{attribute 'GeneratedUsingTerminal: EK1122-0000-0018'}
{attribute addProperty BoxType "EK1122-0000-0018"}
{attribute addProperty Id "Beckhoff_EP2xxxsub_EK1100EK1100_1FC0878B2A_0001_EP2001_1000_0016EP2001_C23D36A611A_0002_EP2001_1000_0017EP2001_C23D36A611A_0003_EP2001_1000_0018EP2001_C23D36A611A_0004_EP2001_1000_0019EP2001_C23D36A611A_0005_EP2008_0001_0016EP2008_E2806B9511A_0006_EP2008_0001_0017EP2008_E2806B9511A_0007_EP2008_0001_0018EP2008_E2806B9511A_0008_EP2008_0001_0019EP2008_E2806B9511A_0009_EP2008_0002_0016EP2008_E2806B9511A_0010_EP2008_0002_0017EP2008_E2806B9511A_0011_EP2008_0002_0018EP2008_E2806B9511A_0012_EP2008_0002_0019EP2008_E2806B9511A_0013_EP2008_0022_0016EP2008_E2806B9511A_0014_EP2008_0022_0017EP2008_E2806B9511A_0015_EP2008_0022_0018EP2008_E2806B9511A_0016_EP2028_0001_0016EP2028_E2806B9511A_0017_EP2028_0001_0017EP2028_E2806B9511A_0018_EP2028_0001_0018EP2028_E2806B9511A_0019_EP2028_0002_0016EP2028_E2806B9511A_0020_EP2028_0002_0017EP2028_E2806B9511A_0021_EP2028_0002_0018EP2028_E2806B9511A_0022_EP2028_0002_0019EP2028_E2806B9511A_0023_EP2028_0032_0017EP2028_E2806B9511A_0024_EP2028_0032_0018EP2028_E2806B9511A_0025_EP2028_0032_0019EP2028_E2806B9511A_0026_EP2038_0001_0016EP2038_3AE10DD720A_0027_EP2038_0001_0017EP2038_3AE10DD720A_0028_EP2038_0001_0018EP2038_3AE10DD720A_0029_EP2038_0002_0016EP2038_3AE10DD720A_0030_EP2038_0002_0017EP2038_3AE10DD720A_0031_EP2038_0002_0018EP2038_3AE10DD720A_0032_EP2308_0000_0016EP2308_F6D9A8D112A_0033_EP2308_0000_0017EP2308_F6D9A8D112A_0034_EP2308_0000_0018EP2308_F6D9A8D112A_0035_EP2308_0001_0016EP2308_F6D9A8D112A_0036_EP2308_0001_0017EP2308_F6D9A8D112A_0037_EP2308_0001_0018EP2308_F6D9A8D112A_0038_EP2308_0001_0019EP2308_F6D9A8D112A_0039_EP2308_0002_0016EP2308_F6D9A8D112A_0040_EP2308_0002_0017EP2308_F6D9A8D112A_0041_EP2308_0002_0018EP2308_F6D9A8D112A_0042_EP2308_0002_0019EP2308_F6D9A8D112A_0043_EP2316_0003_0016EP2316_CAC4656D44A_0044_EP2316_0003_0017EP2316_CAC4656D44A_0045_EP2316_0003_0018EP2316_CAC4656D44A_0046_EP2316_0008_0016EP2316_528F6B1F43A_0047_EP2316_0008_0017EP2316_3C06051444A_0048_EP2316_0008_0018EP2316_DCD24F8F44A_0049_EP2316_0008_0019EP2316_CAC4656D44A_0050_EP2316_0008_0020EP2316_CAC4656D44A_0051_EP2316_0008_0021EP2316_CAC4656D44A_0052_EP2318_0001_0016EP2318_F6D9A8D112A_0053_EP2318_0001_0017EP2318_F6D9A8D112A_0054_EP2318_0001_0018EP2318_F6D9A8D112A_0055_EP2318_0001_0019EP2318_F6D9A8D112A_0056_EP2318_0002_0016EP2318_F6D9A8D112A_0057_EP2318_0002_0017EP2318_F6D9A8D112A_0058_EP2318_0002_0018EP2318_F6D9A8D112A_0059_EP2318_0002_0019EP2318_F6D9A8D112A_0060_EP2328_0001_0016EP2328_F6D9A8D112A_0061_EP2328_0001_0017EP2328_F6D9A8D112A_0062_EP2328_0001_0018EP2328_F6D9A8D112A_0063_EP2328_0002_0016EP2328_F6D9A8D112A_0064_EP2328_0002_0017EP2328_F6D9A8D112A_0065_EP2328_0002_0018EP2328_F6D9A8D112A_0066_EP2328_0002_0019EP2328_F6D9A8D112A_0067_EP2328_1061_0016EP2328_F66CDDB712A_0068_EP2338_0001_0016EP2338_39FFBC5220A_0069_EP2338_0001_0017EP2338_39FFBC5220A_0070_EP2338_0001_0018EP2338_7699BCF620A_0071_EP2338_0001_0019EP2338_7699BCF620A_0072_EP2338_0001_0020EP2338_7699BCF620A_0073_EP2338_0001_0021EP2338_7699BCF620A_0074_EP2338_0001_0022EP2338_7699BCF620A_0075_EP2338_0001_0023EP2338_7699BCF620A_0076_EP2338_0002_0016EP2338_39FFBC5220A_0077_EP2338_0002_0017EP2338_39FFBC5220A_0078_EP2338_0002_0018EP2338_7699BCF620A_0079_EP2338_0002_0019EP2338_7699BCF620A_0080_EP2338_0002_0020EP2338_7699BCF620A_0081_EP2338_0002_0021EP2338_7699BCF620A_0082_EP2338_0002_0022EP2338_7699BCF620A_0083_EP2338_0002_0023EP2338_7699BCF620A_0084_EP2338_1001_0016EP2338_7699BCF620A_0085_EP2338_1001_0017EP2338_7699BCF620A_0086_EP2338_1001_0018EP2338_7699BCF620A_0087_EP2338_1002_0016EP2338_7699BCF620A_0088_EP2338_1002_0017EP2338_7699BCF620A_0089_EP2338_1002_0018EP2338_7699BCF620A_0090_EP2339_0003_0016EP2339_B2B612E850A_0092_EP2339_0021_0016EP2339_C2A6198C42A_0093_EP2339_0021_0017EP2339_D8E9F29A42A_0094_EP2339_0021_0018EP2339_D8E9F29A42A_0095_EP2339_0021_0019EP2339_4CF33DED36A_0096_EP2339_0021_0020EP2339_4CF33DED36A_0097_EP2339_0022_0016EP2339_56BCD6FB36A_0098_EP2339_0022_0017EP2339_4CF33DED36A_0099_EP2339_0022_0018EP2339_4CF33DED36A_0100_EP2339_0022_0019EP2339_4CF33DED36A_0101_EP2339_0042_0017EP2339_4954150736A_0102_EP2339_0042_0018EP2339_E393383136A_0103_EP2339_0121_0016EP2339_4CF33DED36A_0104_EP2349_0021_0016EP2349_4CF33DED36A_0105_EP2349_0021_0017EP2349_4CF33DED36A_0106_EP2349_0021_0018EP2349_4CF33DED36A_0107_EP2349_0022_0016EP2349_4CF33DED36A_0108_EP2349_0022_0017EP2349_4CF33DED36A_0109_EP2349_0022_0018EP2349_4CF33DED36A_0110_EP2624_0002_0016EP2624_7B64371E7A_0111_EP2624_0002_0017EP2624_7B64371E7A_0112_EP2624_0002_0018EP2624_7B64371E7A_0113_EP2624_0002_0019EP2624_7B64371E7A_0114_EP2809_0021_0016EP2809_2B6483BD19A_0115_EP2809_0021_0017EP2809_2B6483BD19A_0116_EP2809_0021_0018EP2809_2B6483BD19A_0117_EP2809_0022_0016EP2809_2B6483BD19A_0118_EP2809_0022_0017EP2809_2B6483BD19A_0119_EP2809_0022_0018EP2809_2B6483BD19A_0120_EP2809_0042_0017EP2809_7AAF2E7119A_0121_EP2809_0042_0018EP2809_23623E9C19A_0122_EP2816_0003_0016EP2816_F9F6AB8251A_0123_EP2816_0004_0016EP2816_8832413327A_0124_EP2816_0004_0017EP2816_F9F6AB8251A_0125_EP2816_0004_0018EP2816_F9F6AB8251A_0126_EP2816_0008_0016EP2816_0C961E2851A_0127_EP2816_0008_0017EP2816_0C961E2851A_0128_EP2816_0008_0018EP2816_D9B77CAE51A_0129_EP2816_0008_0019EP2816_0129644951A_0130_EP2816_0008_0020EP2816_0129644951A_0131_EP2816_0008_0021EP2816_0129644951A_0132_EP2816_0010_0016EP2816_0C961E2851A_0133_EP2816_0010_0017EP2816_0C961E2851A_0134_EP2816_0010_0018EP2816_D9B77CAE51A_0135_EP2816_0010_0019EP2816_0129644951A_0136_EP2816_0010_0020EP2816_0129644951A_0137_EP2816_0010_0021EP2816_0129644951A_0138_EP2817_0008_0016EP2817_7CB3CE2970A_0139_EP2817_0008_0017EP2817_7CB3CE2970A_0140_EP2817_0008_0018EP2817_7CB3CE2970A_0141_EP2817_0008_0019EP2817_7CB3CE2970"}
{attribute addProperty CRC "1783619839"}
{attribute addProperty Size "3524"}
TYPE Beckhoff_EP2xxxEK1122_6A4FE0FF EXTENDS EK1122_1FC0878B :
STRUCT
	{attribute addProperty Name "Beckhoff_EP2xxxsub_EK1100"}
	{attribute addProperty PreviousPort "Beckhoff EP2xxxEK1122 : D"}
	Beckhoff_EP2xxxsub_EK1100 : EK1100_1FC0878B;
	{attribute addProperty Name "A_0001_EP2001_1000_0016"}
	{attribute addProperty PreviousPort "Beckhoff EP2xxxsub EK1100 : C"}
	A_0001_EP2001_1000_0016 : EP2001_C23D36A6;
	{attribute addProperty Name "A_0002_EP2001_1000_0017"}
	{attribute addProperty PreviousPort "A_0001(EP2001-1000-0016) : B"}
	A_0002_EP2001_1000_0017 : EP2001_C23D36A6;
	{attribute addProperty Name "A_0003_EP2001_1000_0018"}
	{attribute addProperty PreviousPort "A_0002(EP2001-1000-0017) : B"}
	A_0003_EP2001_1000_0018 : EP2001_C23D36A6;
	{attribute addProperty Name "A_0004_EP2001_1000_0019"}
	{attribute addProperty PreviousPort "A_0003(EP2001-1000-0018) : B"}
	A_0004_EP2001_1000_0019 : EP2001_C23D36A6;
	{attribute addProperty Name "A_0005_EP2008_0001_0016"}
	{attribute addProperty PreviousPort "A_0004(EP2001-1000-0019) : B"}
	A_0005_EP2008_0001_0016 : EP2008_E2806B95;
	{attribute addProperty Name "A_0006_EP2008_0001_0017"}
	{attribute addProperty PreviousPort "A_0005(EP2008-0001-0016) : B"}
	A_0006_EP2008_0001_0017 : EP2008_E2806B95;
	{attribute addProperty Name "A_0007_EP2008_0001_0018"}
	{attribute addProperty PreviousPort "A_0006(EP2008-0001-0017) : B"}
	A_0007_EP2008_0001_0018 : EP2008_E2806B95;
	{attribute addProperty Name "A_0008_EP2008_0001_0019"}
	{attribute addProperty PreviousPort "A_0007(EP2008-0001-0018) : B"}
	A_0008_EP2008_0001_0019 : EP2008_E2806B95;
	{attribute addProperty Name "A_0009_EP2008_0002_0016"}
	{attribute addProperty PreviousPort "A_0008(EP2008-0001-0019) : B"}
	A_0009_EP2008_0002_0016 : EP2008_E2806B95;
	{attribute addProperty Name "A_0010_EP2008_0002_0017"}
	{attribute addProperty PreviousPort "A_0009(EP2008-0002-0016) : B"}
	A_0010_EP2008_0002_0017 : EP2008_E2806B95;
	{attribute addProperty Name "A_0011_EP2008_0002_0018"}
	{attribute addProperty PreviousPort "A_0010(EP2008-0002-0017) : B"}
	A_0011_EP2008_0002_0018 : EP2008_E2806B95;
	{attribute addProperty Name "A_0012_EP2008_0002_0019"}
	{attribute addProperty PreviousPort "A_0011(EP2008-0002-0018) : B"}
	A_0012_EP2008_0002_0019 : EP2008_E2806B95;
	{attribute addProperty Name "A_0013_EP2008_0022_0016"}
	{attribute addProperty PreviousPort "A_0012(EP2008-0002-0019) : B"}
	A_0013_EP2008_0022_0016 : EP2008_E2806B95;
	{attribute addProperty Name "A_0014_EP2008_0022_0017"}
	{attribute addProperty PreviousPort "A_0013(EP2008-0022-0016) : B"}
	A_0014_EP2008_0022_0017 : EP2008_E2806B95;
	{attribute addProperty Name "A_0015_EP2008_0022_0018"}
	{attribute addProperty PreviousPort "A_0014(EP2008-0022-0017) : B"}
	A_0015_EP2008_0022_0018 : EP2008_E2806B95;
	{attribute addProperty Name "A_0016_EP2028_0001_0016"}
	{attribute addProperty PreviousPort "A_0015(EP2008-0022-0018) : B"}
	A_0016_EP2028_0001_0016 : EP2028_E2806B95;
	{attribute addProperty Name "A_0017_EP2028_0001_0017"}
	{attribute addProperty PreviousPort "A_0016(EP2028-0001-0016) : B"}
	A_0017_EP2028_0001_0017 : EP2028_E2806B95;
	{attribute addProperty Name "A_0018_EP2028_0001_0018"}
	{attribute addProperty PreviousPort "A_0017(EP2028-0001-0017) : B"}
	A_0018_EP2028_0001_0018 : EP2028_E2806B95;
	{attribute addProperty Name "A_0019_EP2028_0002_0016"}
	{attribute addProperty PreviousPort "A_0018(EP2028-0001-0018) : B"}
	A_0019_EP2028_0002_0016 : EP2028_E2806B95;
	{attribute addProperty Name "A_0020_EP2028_0002_0017"}
	{attribute addProperty PreviousPort "A_0019(EP2028-0002-0016) : B"}
	A_0020_EP2028_0002_0017 : EP2028_E2806B95;
	{attribute addProperty Name "A_0021_EP2028_0002_0018"}
	{attribute addProperty PreviousPort "A_0020(EP2028-0002-0017) : B"}
	A_0021_EP2028_0002_0018 : EP2028_E2806B95;
	{attribute addProperty Name "A_0022_EP2028_0002_0019"}
	{attribute addProperty PreviousPort "A_0021(EP2028-0002-0018) : B"}
	A_0022_EP2028_0002_0019 : EP2028_E2806B95;
	{attribute addProperty Name "A_0023_EP2028_0032_0017"}
	{attribute addProperty PreviousPort "A_0022(EP2028-0002-0019) : B"}
	A_0023_EP2028_0032_0017 : EP2028_E2806B95;
	{attribute addProperty Name "A_0024_EP2028_0032_0018"}
	{attribute addProperty PreviousPort "A_0023(EP2028-0032-0017) : B"}
	A_0024_EP2028_0032_0018 : EP2028_E2806B95;
	{attribute addProperty Name "A_0025_EP2028_0032_0019"}
	{attribute addProperty PreviousPort "A_0024(EP2028-0032-0018) : B"}
	A_0025_EP2028_0032_0019 : EP2028_E2806B95;
	{attribute addProperty Name "A_0026_EP2038_0001_0016"}
	{attribute addProperty PreviousPort "A_0025(EP2028-0032-0019) : B"}
	A_0026_EP2038_0001_0016 : EP2038_3AE10DD7;
	{attribute addProperty Name "A_0027_EP2038_0001_0017"}
	{attribute addProperty PreviousPort "A_0026(EP2038-0001-0016) : B"}
	A_0027_EP2038_0001_0017 : EP2038_3AE10DD7;
	{attribute addProperty Name "A_0028_EP2038_0001_0018"}
	{attribute addProperty PreviousPort "A_0027(EP2038-0001-0017) : B"}
	A_0028_EP2038_0001_0018 : EP2038_3AE10DD7;
	{attribute addProperty Name "A_0029_EP2038_0002_0016"}
	{attribute addProperty PreviousPort "A_0028(EP2038-0001-0018) : B"}
	A_0029_EP2038_0002_0016 : EP2038_3AE10DD7;
	{attribute addProperty Name "A_0030_EP2038_0002_0017"}
	{attribute addProperty PreviousPort "A_0029(EP2038-0002-0016) : B"}
	A_0030_EP2038_0002_0017 : EP2038_3AE10DD7;
	{attribute addProperty Name "A_0031_EP2038_0002_0018"}
	{attribute addProperty PreviousPort "A_0030(EP2038-0002-0017) : B"}
	A_0031_EP2038_0002_0018 : EP2038_3AE10DD7;
	{attribute addProperty Name "A_0032_EP2308_0000_0016"}
	{attribute addProperty PreviousPort "A_0031(EP2038-0002-0018) : B"}
	A_0032_EP2308_0000_0016 : EP2308_F6D9A8D1;
	{attribute addProperty Name "A_0033_EP2308_0000_0017"}
	{attribute addProperty PreviousPort "A_0032(EP2308-0000-0016) : B"}
	A_0033_EP2308_0000_0017 : EP2308_F6D9A8D1;
	{attribute addProperty Name "A_0034_EP2308_0000_0018"}
	{attribute addProperty PreviousPort "A_0033(EP2308-0000-0017) : B"}
	A_0034_EP2308_0000_0018 : EP2308_F6D9A8D1;
	{attribute addProperty Name "A_0035_EP2308_0001_0016"}
	{attribute addProperty PreviousPort "A_0034(EP2308-0000-0018) : B"}
	A_0035_EP2308_0001_0016 : EP2308_F6D9A8D1;
	{attribute addProperty Name "A_0036_EP2308_0001_0017"}
	{attribute addProperty PreviousPort "A_0035(EP2308-0001-0016) : B"}
	A_0036_EP2308_0001_0017 : EP2308_F6D9A8D1;
	{attribute addProperty Name "A_0037_EP2308_0001_0018"}
	{attribute addProperty PreviousPort "A_0036(EP2308-0001-0017) : B"}
	A_0037_EP2308_0001_0018 : EP2308_F6D9A8D1;
	{attribute addProperty Name "A_0038_EP2308_0001_0019"}
	{attribute addProperty PreviousPort "A_0037(EP2308-0001-0018) : B"}
	A_0038_EP2308_0001_0019 : EP2308_F6D9A8D1;
	{attribute addProperty Name "A_0039_EP2308_0002_0016"}
	{attribute addProperty PreviousPort "A_0038(EP2308-0001-0019) : B"}
	A_0039_EP2308_0002_0016 : EP2308_F6D9A8D1;
	{attribute addProperty Name "A_0040_EP2308_0002_0017"}
	{attribute addProperty PreviousPort "A_0039(EP2308-0002-0016) : B"}
	A_0040_EP2308_0002_0017 : EP2308_F6D9A8D1;
	{attribute addProperty Name "A_0041_EP2308_0002_0018"}
	{attribute addProperty PreviousPort "A_0040(EP2308-0002-0017) : B"}
	A_0041_EP2308_0002_0018 : EP2308_F6D9A8D1;
	{attribute addProperty Name "A_0042_EP2308_0002_0019"}
	{attribute addProperty PreviousPort "A_0041(EP2308-0002-0018) : B"}
	A_0042_EP2308_0002_0019 : EP2308_F6D9A8D1;
	{attribute addProperty Name "A_0043_EP2316_0003_0016"}
	{attribute addProperty PreviousPort "A_0042(EP2308-0002-0019) : B"}
	A_0043_EP2316_0003_0016 : EP2316_CAC4656D;
	{attribute addProperty Name "A_0044_EP2316_0003_0017"}
	{attribute addProperty PreviousPort "A_0043(EP2316-0003-0016) : B"}
	A_0044_EP2316_0003_0017 : EP2316_CAC4656D;
	{attribute addProperty Name "A_0045_EP2316_0003_0018"}
	{attribute addProperty PreviousPort "A_0044(EP2316-0003-0017) : B"}
	A_0045_EP2316_0003_0018 : EP2316_CAC4656D;
	{attribute addProperty Name "A_0046_EP2316_0008_0016"}
	{attribute addProperty PreviousPort "A_0045(EP2316-0003-0018) : B"}
	A_0046_EP2316_0008_0016 : EP2316_528F6B1F;
	{attribute addProperty Name "A_0047_EP2316_0008_0017"}
	{attribute addProperty PreviousPort "A_0046(EP2316-0008-0016) : B"}
	A_0047_EP2316_0008_0017 : EP2316_3C060514;
	{attribute addProperty Name "A_0048_EP2316_0008_0018"}
	{attribute addProperty PreviousPort "A_0047(EP2316-0008-0017) : B"}
	A_0048_EP2316_0008_0018 : EP2316_DCD24F8F;
	{attribute addProperty Name "A_0049_EP2316_0008_0019"}
	{attribute addProperty PreviousPort "A_0048(EP2316-0008-0018) : B"}
	A_0049_EP2316_0008_0019 : EP2316_CAC4656D;
	{attribute addProperty Name "A_0050_EP2316_0008_0020"}
	{attribute addProperty PreviousPort "A_0049(EP2316-0008-0019) : B"}
	A_0050_EP2316_0008_0020 : EP2316_CAC4656D;
	{attribute addProperty Name "A_0051_EP2316_0008_0021"}
	{attribute addProperty PreviousPort "A_0050(EP2316-0008-0020) : B"}
	A_0051_EP2316_0008_0021 : EP2316_CAC4656D;
	{attribute addProperty Name "A_0052_EP2318_0001_0016"}
	{attribute addProperty PreviousPort "A_0051(EP2316-0008-0021) : B"}
	A_0052_EP2318_0001_0016 : EP2318_F6D9A8D1;
	{attribute addProperty Name "A_0053_EP2318_0001_0017"}
	{attribute addProperty PreviousPort "A_0052(EP2318-0001-0016) : B"}
	A_0053_EP2318_0001_0017 : EP2318_F6D9A8D1;
	{attribute addProperty Name "A_0054_EP2318_0001_0018"}
	{attribute addProperty PreviousPort "A_0053(EP2318-0001-0017) : B"}
	A_0054_EP2318_0001_0018 : EP2318_F6D9A8D1;
	{attribute addProperty Name "A_0055_EP2318_0001_0019"}
	{attribute addProperty PreviousPort "A_0054(EP2318-0001-0018) : B"}
	A_0055_EP2318_0001_0019 : EP2318_F6D9A8D1;
	{attribute addProperty Name "A_0056_EP2318_0002_0016"}
	{attribute addProperty PreviousPort "A_0055(EP2318-0001-0019) : B"}
	A_0056_EP2318_0002_0016 : EP2318_F6D9A8D1;
	{attribute addProperty Name "A_0057_EP2318_0002_0017"}
	{attribute addProperty PreviousPort "A_0056(EP2318-0002-0016) : B"}
	A_0057_EP2318_0002_0017 : EP2318_F6D9A8D1;
	{attribute addProperty Name "A_0058_EP2318_0002_0018"}
	{attribute addProperty PreviousPort "A_0057(EP2318-0002-0017) : B"}
	A_0058_EP2318_0002_0018 : EP2318_F6D9A8D1;
	{attribute addProperty Name "A_0059_EP2318_0002_0019"}
	{attribute addProperty PreviousPort "A_0058(EP2318-0002-0018) : B"}
	A_0059_EP2318_0002_0019 : EP2318_F6D9A8D1;
	{attribute addProperty Name "A_0060_EP2328_0001_0016"}
	{attribute addProperty PreviousPort "A_0059(EP2318-0002-0019) : B"}
	A_0060_EP2328_0001_0016 : EP2328_F6D9A8D1;
	{attribute addProperty Name "A_0061_EP2328_0001_0017"}
	{attribute addProperty PreviousPort "A_0060(EP2328-0001-0016) : B"}
	A_0061_EP2328_0001_0017 : EP2328_F6D9A8D1;
	{attribute addProperty Name "A_0062_EP2328_0001_0018"}
	{attribute addProperty PreviousPort "A_0061(EP2328-0001-0017) : B"}
	A_0062_EP2328_0001_0018 : EP2328_F6D9A8D1;
	{attribute addProperty Name "A_0063_EP2328_0002_0016"}
	{attribute addProperty PreviousPort "A_0062(EP2328-0001-0018) : B"}
	A_0063_EP2328_0002_0016 : EP2328_F6D9A8D1;
	{attribute addProperty Name "A_0064_EP2328_0002_0017"}
	{attribute addProperty PreviousPort "A_0063(EP2328-0002-0016) : B"}
	A_0064_EP2328_0002_0017 : EP2328_F6D9A8D1;
	{attribute addProperty Name "A_0065_EP2328_0002_0018"}
	{attribute addProperty PreviousPort "A_0064(EP2328-0002-0017) : B"}
	A_0065_EP2328_0002_0018 : EP2328_F6D9A8D1;
	{attribute addProperty Name "A_0066_EP2328_0002_0019"}
	{attribute addProperty PreviousPort "A_0065(EP2328-0002-0018) : B"}
	A_0066_EP2328_0002_0019 : EP2328_F6D9A8D1;
	{attribute addProperty Name "A_0067_EP2328_1061_0016"}
	{attribute addProperty PreviousPort "A_0066(EP2328-0002-0019) : B"}
	A_0067_EP2328_1061_0016 : EP2328_F66CDDB7;
	{attribute addProperty Name "A_0068_EP2338_0001_0016"}
	{attribute addProperty PreviousPort "A_0067(EP2328-1061-0016) : B"}
	A_0068_EP2338_0001_0016 : EP2338_39FFBC52;
	{attribute addProperty Name "A_0069_EP2338_0001_0017"}
	{attribute addProperty PreviousPort "A_0068(EP2338-0001-0016) : B"}
	A_0069_EP2338_0001_0017 : EP2338_39FFBC52;
	{attribute addProperty Name "A_0070_EP2338_0001_0018"}
	{attribute addProperty PreviousPort "A_0069(EP2338-0001-0017) : B"}
	A_0070_EP2338_0001_0018 : EP2338_7699BCF6;
	{attribute addProperty Name "A_0071_EP2338_0001_0019"}
	{attribute addProperty PreviousPort "A_0070(EP2338-0001-0018) : B"}
	A_0071_EP2338_0001_0019 : EP2338_7699BCF6;
	{attribute addProperty Name "A_0072_EP2338_0001_0020"}
	{attribute addProperty PreviousPort "A_0071(EP2338-0001-0019) : B"}
	A_0072_EP2338_0001_0020 : EP2338_7699BCF6;
	{attribute addProperty Name "A_0073_EP2338_0001_0021"}
	{attribute addProperty PreviousPort "A_0072(EP2338-0001-0020) : B"}
	A_0073_EP2338_0001_0021 : EP2338_7699BCF6;
	{attribute addProperty Name "A_0074_EP2338_0001_0022"}
	{attribute addProperty PreviousPort "A_0073(EP2338-0001-0021) : B"}
	A_0074_EP2338_0001_0022 : EP2338_7699BCF6;
	{attribute addProperty Name "A_0075_EP2338_0001_0023"}
	{attribute addProperty PreviousPort "A_0074(EP2338-0001-0022) : B"}
	A_0075_EP2338_0001_0023 : EP2338_7699BCF6;
	{attribute addProperty Name "A_0076_EP2338_0002_0016"}
	{attribute addProperty PreviousPort "A_0075(EP2338-0001-0023) : B"}
	A_0076_EP2338_0002_0016 : EP2338_39FFBC52;
	{attribute addProperty Name "A_0077_EP2338_0002_0017"}
	{attribute addProperty PreviousPort "A_0076(EP2338-0002-0016) : B"}
	A_0077_EP2338_0002_0017 : EP2338_39FFBC52;
	{attribute addProperty Name "A_0078_EP2338_0002_0018"}
	{attribute addProperty PreviousPort "A_0077(EP2338-0002-0017) : B"}
	A_0078_EP2338_0002_0018 : EP2338_7699BCF6;
	{attribute addProperty Name "A_0079_EP2338_0002_0019"}
	{attribute addProperty PreviousPort "A_0078(EP2338-0002-0018) : B"}
	A_0079_EP2338_0002_0019 : EP2338_7699BCF6;
	{attribute addProperty Name "A_0080_EP2338_0002_0020"}
	{attribute addProperty PreviousPort "A_0079(EP2338-0002-0019) : B"}
	A_0080_EP2338_0002_0020 : EP2338_7699BCF6;
	{attribute addProperty Name "A_0081_EP2338_0002_0021"}
	{attribute addProperty PreviousPort "A_0080(EP2338-0002-0020) : B"}
	A_0081_EP2338_0002_0021 : EP2338_7699BCF6;
	{attribute addProperty Name "A_0082_EP2338_0002_0022"}
	{attribute addProperty PreviousPort "A_0081(EP2338-0002-0021) : B"}
	A_0082_EP2338_0002_0022 : EP2338_7699BCF6;
	{attribute addProperty Name "A_0083_EP2338_0002_0023"}
	{attribute addProperty PreviousPort "A_0082(EP2338-0002-0022) : B"}
	A_0083_EP2338_0002_0023 : EP2338_7699BCF6;
	{attribute addProperty Name "A_0084_EP2338_1001_0016"}
	{attribute addProperty PreviousPort "A_0083(EP2338-0002-0023) : B"}
	A_0084_EP2338_1001_0016 : EP2338_7699BCF6;
	{attribute addProperty Name "A_0085_EP2338_1001_0017"}
	{attribute addProperty PreviousPort "A_0084(EP2338-1001-0016) : B"}
	A_0085_EP2338_1001_0017 : EP2338_7699BCF6;
	{attribute addProperty Name "A_0086_EP2338_1001_0018"}
	{attribute addProperty PreviousPort "A_0085(EP2338-1001-0017) : B"}
	A_0086_EP2338_1001_0018 : EP2338_7699BCF6;
	{attribute addProperty Name "A_0087_EP2338_1002_0016"}
	{attribute addProperty PreviousPort "A_0086(EP2338-1001-0018) : B"}
	A_0087_EP2338_1002_0016 : EP2338_7699BCF6;
	{attribute addProperty Name "A_0088_EP2338_1002_0017"}
	{attribute addProperty PreviousPort "A_0087(EP2338-1002-0016) : B"}
	A_0088_EP2338_1002_0017 : EP2338_7699BCF6;
	{attribute addProperty Name "A_0089_EP2338_1002_0018"}
	{attribute addProperty PreviousPort "A_0088(EP2338-1002-0017) : B"}
	A_0089_EP2338_1002_0018 : EP2338_7699BCF6;
	{attribute addProperty Name "A_0090_EP2339_0003_0016"}
	{attribute addProperty PreviousPort "A_0089(EP2338-1002-0018) : B"}
	A_0090_EP2339_0003_0016 : EP2339_B2B612E8;
	{attribute addProperty Name "A_0092_EP2339_0021_0016"}
	{attribute addProperty PreviousPort "A_0090(EP2339-0003-0016) : B"}
	A_0092_EP2339_0021_0016 : EP2339_C2A6198C;
	{attribute addProperty Name "A_0093_EP2339_0021_0017"}
	{attribute addProperty PreviousPort "A_0092(EP2339-0021-0016) : B"}
	A_0093_EP2339_0021_0017 : EP2339_D8E9F29A;
	{attribute addProperty Name "A_0094_EP2339_0021_0018"}
	{attribute addProperty PreviousPort "A_0093(EP2339-0021-0017) : B"}
	A_0094_EP2339_0021_0018 : EP2339_D8E9F29A;
	{attribute addProperty Name "A_0095_EP2339_0021_0019"}
	{attribute addProperty PreviousPort "A_0094(EP2339-0021-0018) : B"}
	A_0095_EP2339_0021_0019 : EP2339_4CF33DED;
	{attribute addProperty Name "A_0096_EP2339_0021_0020"}
	{attribute addProperty PreviousPort "A_0095(EP2339-0021-0019) : B"}
	A_0096_EP2339_0021_0020 : EP2339_4CF33DED;
	{attribute addProperty Name "A_0097_EP2339_0022_0016"}
	{attribute addProperty PreviousPort "A_0096(EP2339-0021-0020) : B"}
	A_0097_EP2339_0022_0016 : EP2339_56BCD6FB;
	{attribute addProperty Name "A_0098_EP2339_0022_0017"}
	{attribute addProperty PreviousPort "A_0097(EP2339-0022-0016) : B"}
	A_0098_EP2339_0022_0017 : EP2339_4CF33DED;
	{attribute addProperty Name "A_0099_EP2339_0022_0018"}
	{attribute addProperty PreviousPort "A_0098(EP2339-0022-0017) : B"}
	A_0099_EP2339_0022_0018 : EP2339_4CF33DED;
	{attribute addProperty Name "A_0100_EP2339_0022_0019"}
	{attribute addProperty PreviousPort "A_0099(EP2339-0022-0018) : B"}
	A_0100_EP2339_0022_0019 : EP2339_4CF33DED;
	{attribute addProperty Name "A_0101_EP2339_0042_0017"}
	{attribute addProperty PreviousPort "A_0100(EP2339-0022-0019) : B"}
	A_0101_EP2339_0042_0017 : EP2339_49541507;
	{attribute addProperty Name "A_0102_EP2339_0042_0018"}
	{attribute addProperty PreviousPort "A_0101(EP2339-0042-0017) : B"}
	A_0102_EP2339_0042_0018 : EP2339_E3933831;
	{attribute addProperty Name "A_0103_EP2339_0121_0016"}
	{attribute addProperty PreviousPort "A_0102(EP2339-0042-0018) : B"}
	A_0103_EP2339_0121_0016 : EP2339_4CF33DED;
	{attribute addProperty Name "A_0104_EP2349_0021_0016"}
	{attribute addProperty PreviousPort "A_0103(EP2339-0121-0016) : B"}
	A_0104_EP2349_0021_0016 : EP2349_4CF33DED;
	{attribute addProperty Name "A_0105_EP2349_0021_0017"}
	{attribute addProperty PreviousPort "A_0104(EP2349-0021-0016) : B"}
	A_0105_EP2349_0021_0017 : EP2349_4CF33DED;
	{attribute addProperty Name "A_0106_EP2349_0021_0018"}
	{attribute addProperty PreviousPort "A_0105(EP2349-0021-0017) : B"}
	A_0106_EP2349_0021_0018 : EP2349_4CF33DED;
	{attribute addProperty Name "A_0107_EP2349_0022_0016"}
	{attribute addProperty PreviousPort "A_0106(EP2349-0021-0018) : B"}
	A_0107_EP2349_0022_0016 : EP2349_4CF33DED;
	{attribute addProperty Name "A_0108_EP2349_0022_0017"}
	{attribute addProperty PreviousPort "A_0107(EP2349-0022-0016) : B"}
	A_0108_EP2349_0022_0017 : EP2349_4CF33DED;
	{attribute addProperty Name "A_0109_EP2349_0022_0018"}
	{attribute addProperty PreviousPort "A_0108(EP2349-0022-0017) : B"}
	A_0109_EP2349_0022_0018 : EP2349_4CF33DED;
	{attribute addProperty Name "A_0110_EP2624_0002_0016"}
	{attribute addProperty PreviousPort "A_0109(EP2349-0022-0018) : B"}
	A_0110_EP2624_0002_0016 : EP2624_7B64371E;
	{attribute addProperty Name "A_0111_EP2624_0002_0017"}
	{attribute addProperty PreviousPort "A_0110(EP2624-0002-0016) : B"}
	A_0111_EP2624_0002_0017 : EP2624_7B64371E;
	{attribute addProperty Name "A_0112_EP2624_0002_0018"}
	{attribute addProperty PreviousPort "A_0111(EP2624-0002-0017) : B"}
	A_0112_EP2624_0002_0018 : EP2624_7B64371E;
	{attribute addProperty Name "A_0113_EP2624_0002_0019"}
	{attribute addProperty PreviousPort "A_0112(EP2624-0002-0018) : B"}
	A_0113_EP2624_0002_0019 : EP2624_7B64371E;
	{attribute addProperty Name "A_0114_EP2809_0021_0016"}
	{attribute addProperty PreviousPort "A_0113(EP2624-0002-0019) : B"}
	A_0114_EP2809_0021_0016 : EP2809_2B6483BD;
	{attribute addProperty Name "A_0115_EP2809_0021_0017"}
	{attribute addProperty PreviousPort "A_0114(EP2809-0021-0016) : B"}
	A_0115_EP2809_0021_0017 : EP2809_2B6483BD;
	{attribute addProperty Name "A_0116_EP2809_0021_0018"}
	{attribute addProperty PreviousPort "A_0115(EP2809-0021-0017) : B"}
	A_0116_EP2809_0021_0018 : EP2809_2B6483BD;
	{attribute addProperty Name "A_0117_EP2809_0022_0016"}
	{attribute addProperty PreviousPort "A_0116(EP2809-0021-0018) : B"}
	A_0117_EP2809_0022_0016 : EP2809_2B6483BD;
	{attribute addProperty Name "A_0118_EP2809_0022_0017"}
	{attribute addProperty PreviousPort "A_0117(EP2809-0022-0016) : B"}
	A_0118_EP2809_0022_0017 : EP2809_2B6483BD;
	{attribute addProperty Name "A_0119_EP2809_0022_0018"}
	{attribute addProperty PreviousPort "A_0118(EP2809-0022-0017) : B"}
	A_0119_EP2809_0022_0018 : EP2809_2B6483BD;
	{attribute addProperty Name "A_0120_EP2809_0042_0017"}
	{attribute addProperty PreviousPort "A_0119(EP2809-0022-0018) : B"}
	A_0120_EP2809_0042_0017 : EP2809_7AAF2E71;
	{attribute addProperty Name "A_0121_EP2809_0042_0018"}
	{attribute addProperty PreviousPort "A_0120(EP2809-0042-0017) : B"}
	A_0121_EP2809_0042_0018 : EP2809_23623E9C;
	{attribute addProperty Name "A_0122_EP2816_0003_0016"}
	{attribute addProperty PreviousPort "A_0121(EP2809-0042-0018) : B"}
	A_0122_EP2816_0003_0016 : EP2816_F9F6AB82;
	{attribute addProperty Name "A_0123_EP2816_0004_0016"}
	{attribute addProperty PreviousPort "A_0122(EP2816-0003-0016) : B"}
	A_0123_EP2816_0004_0016 : EP2816_88324133;
	{attribute addProperty Name "A_0124_EP2816_0004_0017"}
	{attribute addProperty PreviousPort "A_0123(EP2816-0004-0016) : B"}
	A_0124_EP2816_0004_0017 : EP2816_F9F6AB82;
	{attribute addProperty Name "A_0125_EP2816_0004_0018"}
	{attribute addProperty PreviousPort "A_0124(EP2816-0004-0017) : B"}
	A_0125_EP2816_0004_0018 : EP2816_F9F6AB82;
	{attribute addProperty Name "A_0126_EP2816_0008_0016"}
	{attribute addProperty PreviousPort "A_0125(EP2816-0004-0018) : B"}
	A_0126_EP2816_0008_0016 : EP2816_0C961E28;
	{attribute addProperty Name "A_0127_EP2816_0008_0017"}
	{attribute addProperty PreviousPort "A_0126(EP2816-0008-0016) : B"}
	A_0127_EP2816_0008_0017 : EP2816_0C961E28;
	{attribute addProperty Name "A_0128_EP2816_0008_0018"}
	{attribute addProperty PreviousPort "A_0127(EP2816-0008-0017) : B"}
	A_0128_EP2816_0008_0018 : EP2816_D9B77CAE;
	{attribute addProperty Name "A_0129_EP2816_0008_0019"}
	{attribute addProperty PreviousPort "A_0128(EP2816-0008-0018) : B"}
	A_0129_EP2816_0008_0019 : EP2816_01296449;
	{attribute addProperty Name "A_0130_EP2816_0008_0020"}
	{attribute addProperty PreviousPort "A_0129(EP2816-0008-0019) : B"}
	A_0130_EP2816_0008_0020 : EP2816_01296449;
	{attribute addProperty Name "A_0131_EP2816_0008_0021"}
	{attribute addProperty PreviousPort "A_0130(EP2816-0008-0020) : B"}
	A_0131_EP2816_0008_0021 : EP2816_01296449;
	{attribute addProperty Name "A_0132_EP2816_0010_0016"}
	{attribute addProperty PreviousPort "A_0131(EP2816-0008-0021) : B"}
	A_0132_EP2816_0010_0016 : EP2816_0C961E28;
	{attribute addProperty Name "A_0133_EP2816_0010_0017"}
	{attribute addProperty PreviousPort "A_0132(EP2816-0010-0016) : B"}
	A_0133_EP2816_0010_0017 : EP2816_0C961E28;
	{attribute addProperty Name "A_0134_EP2816_0010_0018"}
	{attribute addProperty PreviousPort "A_0133(EP2816-0010-0017) : B"}
	A_0134_EP2816_0010_0018 : EP2816_D9B77CAE;
	{attribute addProperty Name "A_0135_EP2816_0010_0019"}
	{attribute addProperty PreviousPort "A_0134(EP2816-0010-0018) : B"}
	A_0135_EP2816_0010_0019 : EP2816_01296449;
	{attribute addProperty Name "A_0136_EP2816_0010_0020"}
	{attribute addProperty PreviousPort "A_0135(EP2816-0010-0019) : B"}
	A_0136_EP2816_0010_0020 : EP2816_01296449;
	{attribute addProperty Name "A_0137_EP2816_0010_0021"}
	{attribute addProperty PreviousPort "A_0136(EP2816-0010-0020) : B"}
	A_0137_EP2816_0010_0021 : EP2816_01296449;
	{attribute addProperty Name "A_0138_EP2817_0008_0016"}
	{attribute addProperty PreviousPort "A_0137(EP2816-0010-0021) : B"}
	A_0138_EP2817_0008_0016 : EP2817_7CB3CE29;
	{attribute addProperty Name "A_0139_EP2817_0008_0017"}
	{attribute addProperty PreviousPort "A_0138(EP2817-0008-0016) : B"}
	A_0139_EP2817_0008_0017 : EP2817_7CB3CE29;
	{attribute addProperty Name "A_0140_EP2817_0008_0018"}
	{attribute addProperty PreviousPort "A_0139(EP2817-0008-0017) : B"}
	A_0140_EP2817_0008_0018 : EP2817_7CB3CE29;
	{attribute addProperty Name "A_0141_EP2817_0008_0019"}
	{attribute addProperty PreviousPort "A_0140(EP2817-0008-0018) : B"}
	A_0141_EP2817_0008_0019 : EP2817_7CB3CE29;
END_STRUCT
END_TYPE

(* stored: Version 1.2.0.0, ProductVersion 3.1.4024.9
   DUT Beckhoff_EP2xxxEK1122_6A4FE0FF: Id {f4047407-1b19-4590-b435-c644c44ea369} *)
